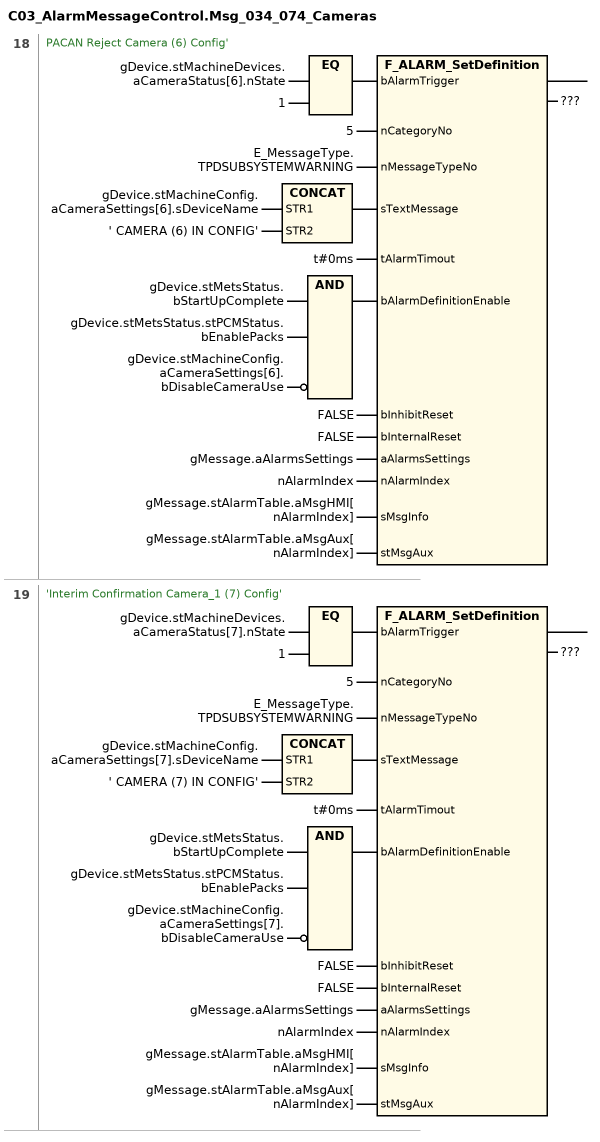
// NETWORK 18
// PACAN Reject Camera (6) Config'
F_ALARM_SetDefinition(bAlarmTrigger := gDevice.stMachineDevices.aCameraStatus[6].nState = 1, nCategoryNo := 5, nMessageTypeNo := E_MessageType.TPDSUBSYSTEMWARNING, sTextMessage := CONCAT(STR1 := gDevice.stMachineConfig.aCameraSettings[6].sDeviceName, STR2 := ' CAMERA (6) IN CONFIG'), tAlarmTimout := t#0ms, bAlarmDefinitionEnable := gDevice.stMetsStatus.bStartUpComplete AND gDevice.stMetsStatus.stPCMStatus.bEnablePacks AND NOT gDevice.stMachineConfig.aCameraSettings[6].bDisableCameraUse, bInhibitReset := FALSE, bInternalReset := FALSE, aAlarmsSettings := gMessage.aAlarmsSettings, nAlarmIndex := nAlarmIndex, sMsgInfo := gMessage.stAlarmTable.aMsgHMI[nAlarmIndex], stMsgAux := gMessage.stAlarmTable.aMsgAux[nAlarmIndex]);

// NETWORK 19
// 'Interim Confirmation Camera_1 (7) Config'
F_ALARM_SetDefinition(bAlarmTrigger := gDevice.stMachineDevices.aCameraStatus[7].nState = 1, nCategoryNo := 5, nMessageTypeNo := E_MessageType.TPDSUBSYSTEMWARNING, sTextMessage := CONCAT(STR1 := gDevice.stMachineConfig.aCameraSettings[7].sDeviceName, STR2 := ' CAMERA (7) IN CONFIG'), tAlarmTimout := t#0ms, bAlarmDefinitionEnable := gDevice.stMetsStatus.bStartUpComplete AND gDevice.stMetsStatus.stPCMStatus.bEnablePacks AND NOT gDevice.stMachineConfig.aCameraSettings[7].bDisableCameraUse, bInhibitReset := FALSE, bInternalReset := FALSE, aAlarmsSettings := gMessage.aAlarmsSettings, nAlarmIndex := nAlarmIndex, sMsgInfo := gMessage.stAlarmTable.aMsgHMI[nAlarmIndex], stMsgAux := gMessage.stAlarmTable.aMsgAux[nAlarmIndex]);

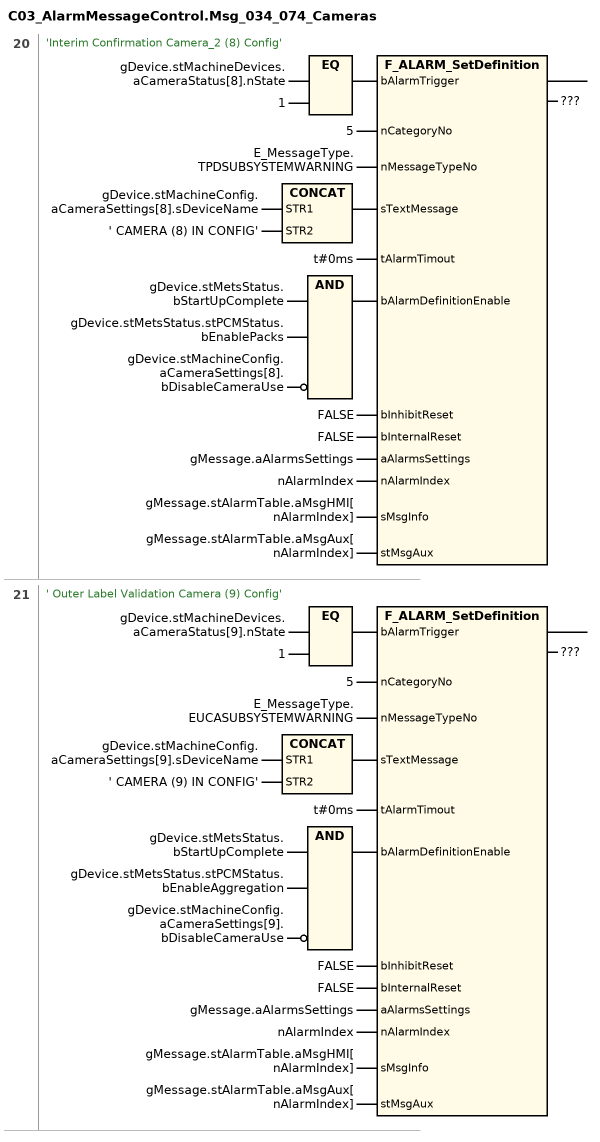
// NETWORK 20
// 'Interim Confirmation Camera_2 (8) Config'
F_ALARM_SetDefinition(bAlarmTrigger := gDevice.stMachineDevices.aCameraStatus[8].nState = 1, nCategoryNo := 5, nMessageTypeNo := E_MessageType.TPDSUBSYSTEMWARNING, sTextMessage := CONCAT(STR1 := gDevice.stMachineConfig.aCameraSettings[8].sDeviceName, STR2 := ' CAMERA (8) IN CONFIG'), tAlarmTimout := t#0ms, bAlarmDefinitionEnable := gDevice.stMetsStatus.bStartUpComplete AND gDevice.stMetsStatus.stPCMStatus.bEnablePacks AND NOT gDevice.stMachineConfig.aCameraSettings[8].bDisableCameraUse, bInhibitReset := FALSE, bInternalReset := FALSE, aAlarmsSettings := gMessage.aAlarmsSettings, nAlarmIndex := nAlarmIndex, sMsgInfo := gMessage.stAlarmTable.aMsgHMI[nAlarmIndex], stMsgAux := gMessage.stAlarmTable.aMsgAux[nAlarmIndex]);

// NETWORK 21
// ' Outer Label Validation Camera (9) Config'
F_ALARM_SetDefinition(bAlarmTrigger := gDevice.stMachineDevices.aCameraStatus[9].nState = 1, nCategoryNo := 5, nMessageTypeNo := E_MessageType.EUCASUBSYSTEMWARNING, sTextMessage := CONCAT(STR1 := gDevice.stMachineConfig.aCameraSettings[9].sDeviceName, STR2 := ' CAMERA (9) IN CONFIG'), tAlarmTimout := t#0ms, bAlarmDefinitionEnable := gDevice.stMetsStatus.bStartUpComplete AND gDevice.stMetsStatus.stPCMStatus.bEnableAggregation AND NOT gDevice.stMachineConfig.aCameraSettings[9].bDisableCameraUse, bInhibitReset := FALSE, bInternalReset := FALSE, aAlarmsSettings := gMessage.aAlarmsSettings, nAlarmIndex := nAlarmIndex, sMsgInfo := gMessage.stAlarmTable.aMsgHMI[nAlarmIndex], stMsgAux := gMessage.stAlarmTable.aMsgAux[nAlarmIndex]);

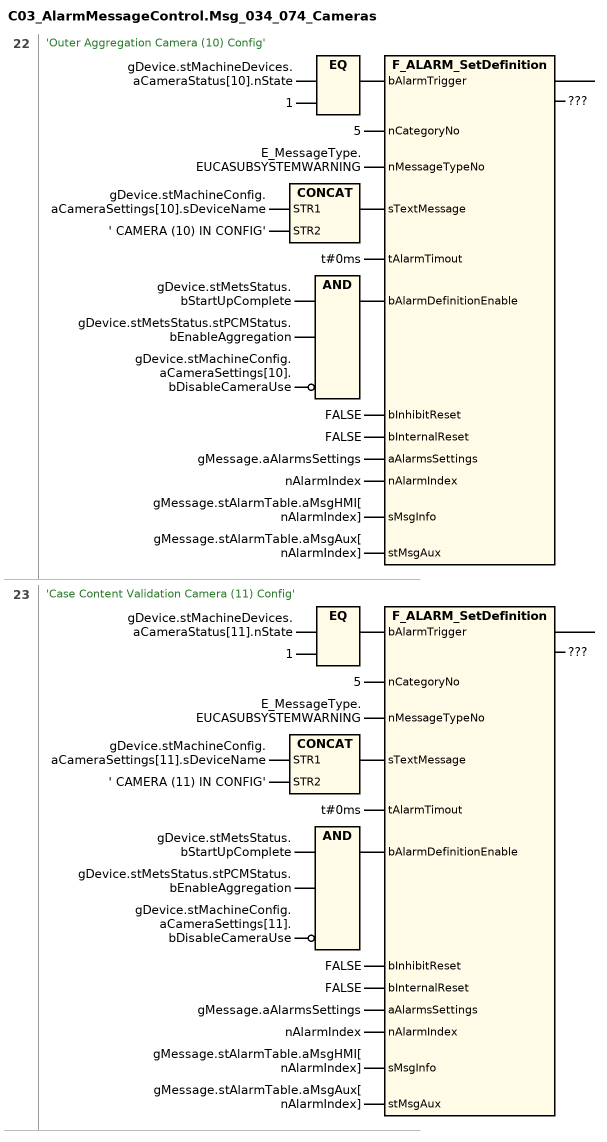
// NETWORK 22
// 'Outer Aggregation Camera (10) Config'
F_ALARM_SetDefinition(bAlarmTrigger := gDevice.stMachineDevices.aCameraStatus[10].nState = 1, nCategoryNo := 5, nMessageTypeNo := E_MessageType.EUCASUBSYSTEMWARNING, sTextMessage := CONCAT(STR1 := gDevice.stMachineConfig.aCameraSettings[10].sDeviceName, STR2 := ' CAMERA (10) IN CONFIG'), tAlarmTimout := t#0ms, bAlarmDefinitionEnable := gDevice.stMetsStatus.bStartUpComplete AND gDevice.stMetsStatus.stPCMStatus.bEnableAggregation AND NOT gDevice.stMachineConfig.aCameraSettings[10].bDisableCameraUse, bInhibitReset := FALSE, bInternalReset := FALSE, aAlarmsSettings := gMessage.aAlarmsSettings, nAlarmIndex := nAlarmIndex, sMsgInfo := gMessage.stAlarmTable.aMsgHMI[nAlarmIndex], stMsgAux := gMessage.stAlarmTable.aMsgAux[nAlarmIndex]);

// NETWORK 23
// 'Case Content Validation Camera (11) Config'
F_ALARM_SetDefinition(bAlarmTrigger := gDevice.stMachineDevices.aCameraStatus[11].nState = 1, nCategoryNo := 5, nMessageTypeNo := E_MessageType.EUCASUBSYSTEMWARNING, sTextMessage := CONCAT(STR1 := gDevice.stMachineConfig.aCameraSettings[11].sDeviceName, STR2 := ' CAMERA (11) IN CONFIG'), tAlarmTimout := t#0ms, bAlarmDefinitionEnable := gDevice.stMetsStatus.bStartUpComplete AND gDevice.stMetsStatus.stPCMStatus.bEnableAggregation AND NOT gDevice.stMachineConfig.aCameraSettings[11].bDisableCameraUse, bInhibitReset := FALSE, bInternalReset := FALSE, aAlarmsSettings := gMessage.aAlarmsSettings, nAlarmIndex := nAlarmIndex, sMsgInfo := gMessage.stAlarmTable.aMsgHMI[nAlarmIndex], stMsgAux := gMessage.stAlarmTable.aMsgAux[nAlarmIndex]);

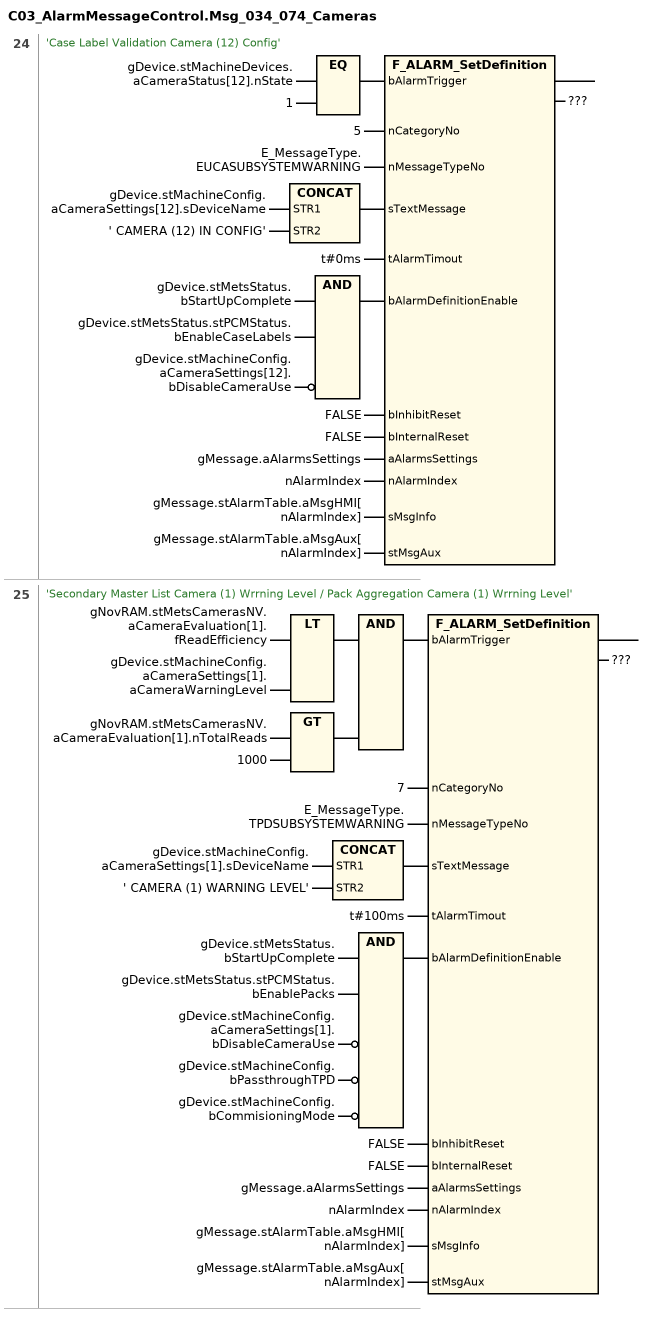
// NETWORK 24
// 'Case Label Validation Camera (12) Config'
F_ALARM_SetDefinition(bAlarmTrigger := gDevice.stMachineDevices.aCameraStatus[12].nState = 1, nCategoryNo := 5, nMessageTypeNo := E_MessageType.EUCASUBSYSTEMWARNING, sTextMessage := CONCAT(STR1 := gDevice.stMachineConfig.aCameraSettings[12].sDeviceName, STR2 := ' CAMERA (12) IN CONFIG'), tAlarmTimout := t#0ms, bAlarmDefinitionEnable := gDevice.stMetsStatus.bStartUpComplete AND gDevice.stMetsStatus.stPCMStatus.bEnableCaseLabels AND NOT gDevice.stMachineConfig.aCameraSettings[12].bDisableCameraUse, bInhibitReset := FALSE, bInternalReset := FALSE, aAlarmsSettings := gMessage.aAlarmsSettings, nAlarmIndex := nAlarmIndex, sMsgInfo := gMessage.stAlarmTable.aMsgHMI[nAlarmIndex], stMsgAux := gMessage.stAlarmTable.aMsgAux[nAlarmIndex]);

// NETWORK 25
// 'Secondary Master List Camera (1) Wrrning Level / Pack Aggregation Camera (1) Wrrning Level'
F_ALARM_SetDefinition(bAlarmTrigger := gNovRAM.stMetsCamerasNV.aCameraEvaluation[1].fReadEfficiency < gDevice.stMachineConfig.aCameraSettings[1].aCameraWarningLevel AND gNovRAM.stMetsCamerasNV.aCameraEvaluation[1].nTotalReads > 1000, nCategoryNo := 7, nMessageTypeNo := E_MessageType.TPDSUBSYSTEMWARNING, sTextMessage := CONCAT(STR1 := gDevice.stMachineConfig.aCameraSettings[1].sDeviceName, STR2 := ' CAMERA (1) WARNING LEVEL'), tAlarmTimout := t#100ms, bAlarmDefinitionEnable := gDevice.stMetsStatus.bStartUpComplete AND gDevice.stMetsStatus.stPCMStatus.bEnablePacks AND NOT gDevice.stMachineConfig.aCameraSettings[1].bDisableCameraUse AND NOT gDevice.stMachineConfig.bPassthroughTPD AND NOT gDevice.stMachineConfig.bCommisioningMode, bInhibitReset := FALSE, bInternalReset := FALSE, aAlarmsSettings := gMessage.aAlarmsSettings, nAlarmIndex := nAlarmIndex, sMsgInfo := gMessage.stAlarmTable.aMsgHMI[nAlarmIndex], stMsgAux := gMessage.stAlarmTable.aMsgAux[nAlarmIndex]);

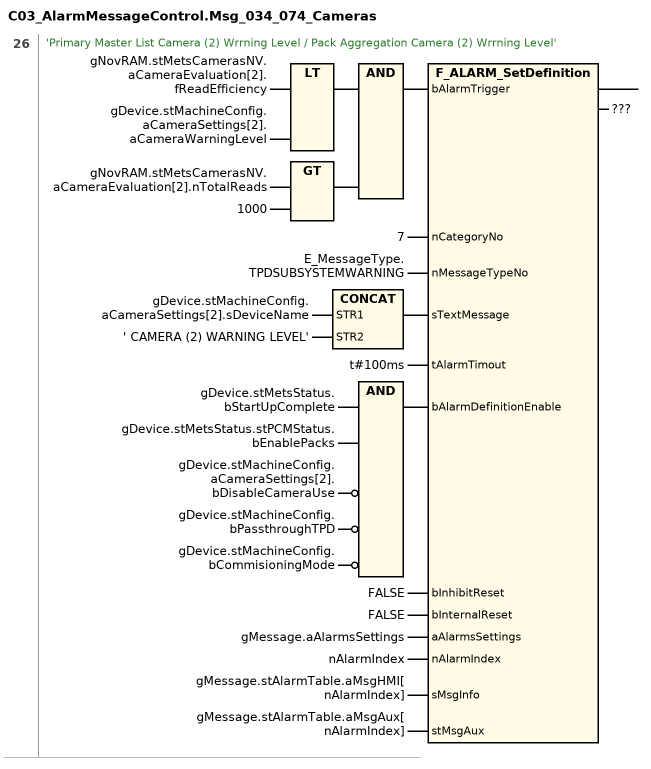
// NETWORK 26
// 'Primary Master List Camera (2) Wrrning Level / Pack Aggregation Camera (2) Wrrning Level'
F_ALARM_SetDefinition(bAlarmTrigger := gNovRAM.stMetsCamerasNV.aCameraEvaluation[2].fReadEfficiency < gDevice.stMachineConfig.aCameraSettings[2].aCameraWarningLevel AND gNovRAM.stMetsCamerasNV.aCameraEvaluation[2].nTotalReads > 1000, nCategoryNo := 7, nMessageTypeNo := E_MessageType.TPDSUBSYSTEMWARNING, sTextMessage := CONCAT(STR1 := gDevice.stMachineConfig.aCameraSettings[2].sDeviceName, STR2 := ' CAMERA (2) WARNING LEVEL'), tAlarmTimout := t#100ms, bAlarmDefinitionEnable := gDevice.stMetsStatus.bStartUpComplete AND gDevice.stMetsStatus.stPCMStatus.bEnablePacks AND NOT gDevice.stMachineConfig.aCameraSettings[2].bDisableCameraUse AND NOT gDevice.stMachineConfig.bPassthroughTPD AND NOT gDevice.stMachineConfig.bCommisioningMode, bInhibitReset := FALSE, bInternalReset := FALSE, aAlarmsSettings := gMessage.aAlarmsSettings, nAlarmIndex := nAlarmIndex, sMsgInfo := gMessage.stAlarmTable.aMsgHMI[nAlarmIndex], stMsgAux := gMessage.stAlarmTable.aMsgAux[nAlarmIndex]);

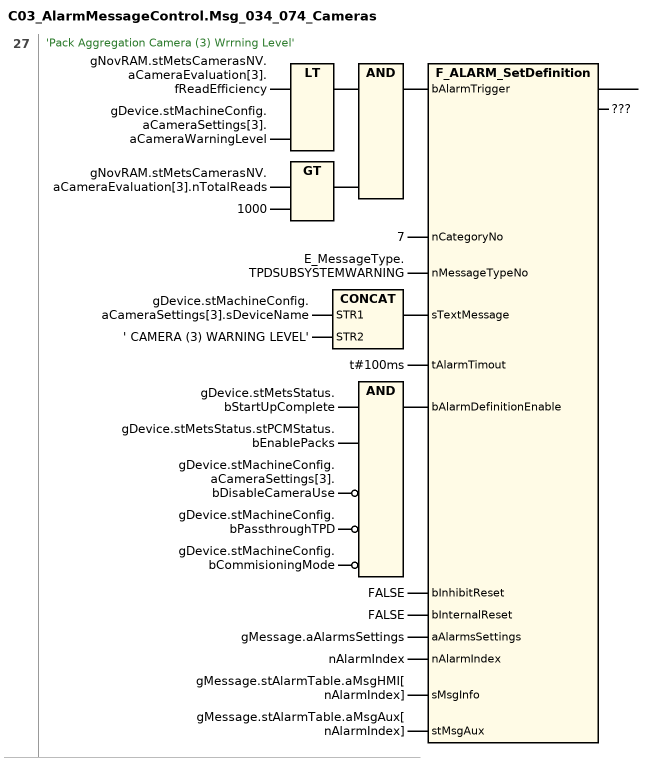
// NETWORK 27
// 'Pack Aggregation Camera (3) Wrrning Level'
F_ALARM_SetDefinition(bAlarmTrigger := gNovRAM.stMetsCamerasNV.aCameraEvaluation[3].fReadEfficiency < gDevice.stMachineConfig.aCameraSettings[3].aCameraWarningLevel AND gNovRAM.stMetsCamerasNV.aCameraEvaluation[3].nTotalReads > 1000, nCategoryNo := 7, nMessageTypeNo := E_MessageType.TPDSUBSYSTEMWARNING, sTextMessage := CONCAT(STR1 := gDevice.stMachineConfig.aCameraSettings[3].sDeviceName, STR2 := ' CAMERA (3) WARNING LEVEL'), tAlarmTimout := t#100ms, bAlarmDefinitionEnable := gDevice.stMetsStatus.bStartUpComplete AND gDevice.stMetsStatus.stPCMStatus.bEnablePacks AND NOT gDevice.stMachineConfig.aCameraSettings[3].bDisableCameraUse AND NOT gDevice.stMachineConfig.bPassthroughTPD AND NOT gDevice.stMachineConfig.bCommisioningMode, bInhibitReset := FALSE, bInternalReset := FALSE, aAlarmsSettings := gMessage.aAlarmsSettings, nAlarmIndex := nAlarmIndex, sMsgInfo := gMessage.stAlarmTable.aMsgHMI[nAlarmIndex], stMsgAux := gMessage.stAlarmTable.aMsgAux[nAlarmIndex]);

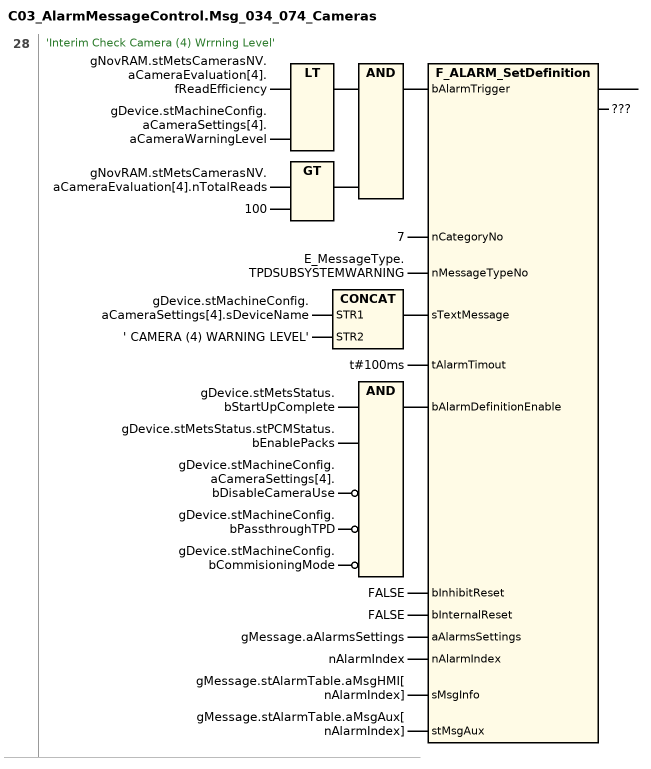
// NETWORK 28
// 'Interim Check Camera (4) Wrrning Level'
F_ALARM_SetDefinition(bAlarmTrigger := gNovRAM.stMetsCamerasNV.aCameraEvaluation[4].fReadEfficiency < gDevice.stMachineConfig.aCameraSettings[4].aCameraWarningLevel AND gNovRAM.stMetsCamerasNV.aCameraEvaluation[4].nTotalReads > 100, nCategoryNo := 7, nMessageTypeNo := E_MessageType.TPDSUBSYSTEMWARNING, sTextMessage := CONCAT(STR1 := gDevice.stMachineConfig.aCameraSettings[4].sDeviceName, STR2 := ' CAMERA (4) WARNING LEVEL'), tAlarmTimout := t#100ms, bAlarmDefinitionEnable := gDevice.stMetsStatus.bStartUpComplete AND gDevice.stMetsStatus.stPCMStatus.bEnablePacks AND NOT gDevice.stMachineConfig.aCameraSettings[4].bDisableCameraUse AND NOT gDevice.stMachineConfig.bPassthroughTPD AND NOT gDevice.stMachineConfig.bCommisioningMode, bInhibitReset := FALSE, bInternalReset := FALSE, aAlarmsSettings := gMessage.aAlarmsSettings, nAlarmIndex := nAlarmIndex, sMsgInfo := gMessage.stAlarmTable.aMsgHMI[nAlarmIndex], stMsgAux := gMessage.stAlarmTable.aMsgAux[nAlarmIndex]);

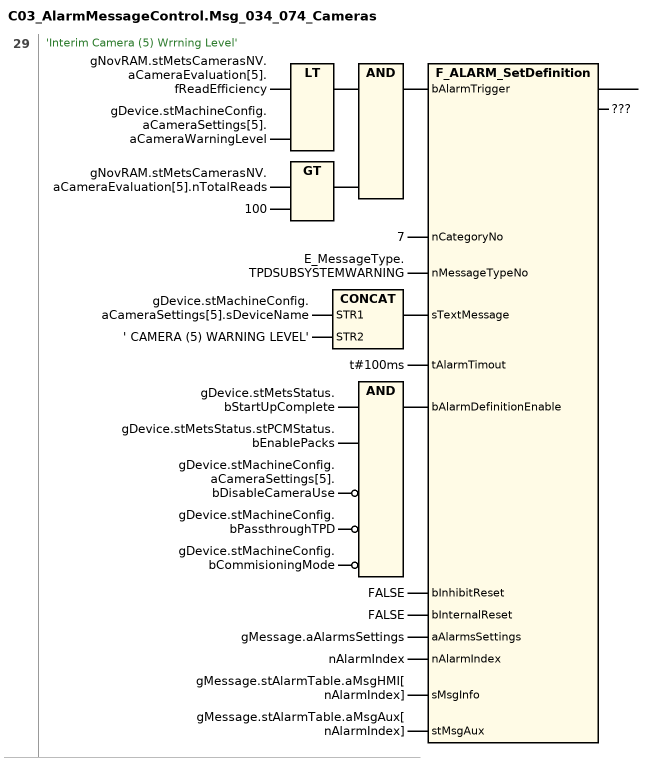
// NETWORK 29
// 'Interim Camera (5) Wrrning Level'
F_ALARM_SetDefinition(bAlarmTrigger := gNovRAM.stMetsCamerasNV.aCameraEvaluation[5].fReadEfficiency < gDevice.stMachineConfig.aCameraSettings[5].aCameraWarningLevel AND gNovRAM.stMetsCamerasNV.aCameraEvaluation[5].nTotalReads > 100, nCategoryNo := 7, nMessageTypeNo := E_MessageType.TPDSUBSYSTEMWARNING, sTextMessage := CONCAT(STR1 := gDevice.stMachineConfig.aCameraSettings[5].sDeviceName, STR2 := ' CAMERA (5) WARNING LEVEL'), tAlarmTimout := t#100ms, bAlarmDefinitionEnable := gDevice.stMetsStatus.bStartUpComplete AND gDevice.stMetsStatus.stPCMStatus.bEnablePacks AND NOT gDevice.stMachineConfig.aCameraSettings[5].bDisableCameraUse AND NOT gDevice.stMachineConfig.bPassthroughTPD AND NOT gDevice.stMachineConfig.bCommisioningMode, bInhibitReset := FALSE, bInternalReset := FALSE, aAlarmsSettings := gMessage.aAlarmsSettings, nAlarmIndex := nAlarmIndex, sMsgInfo := gMessage.stAlarmTable.aMsgHMI[nAlarmIndex], stMsgAux := gMessage.stAlarmTable.aMsgAux[nAlarmIndex]);

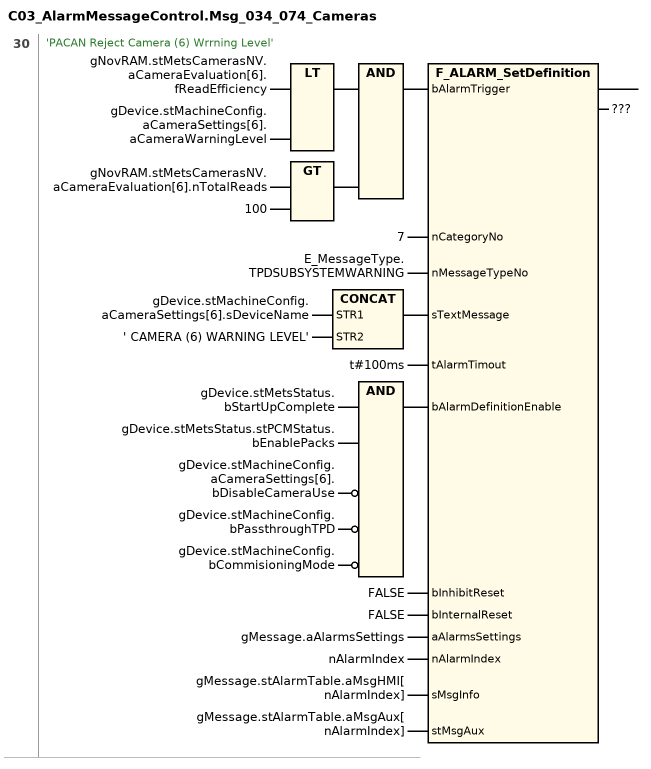
// NETWORK 30
// 'PACAN Reject Camera (6) Wrrning Level'
F_ALARM_SetDefinition(bAlarmTrigger := gNovRAM.stMetsCamerasNV.aCameraEvaluation[6].fReadEfficiency < gDevice.stMachineConfig.aCameraSettings[6].aCameraWarningLevel AND gNovRAM.stMetsCamerasNV.aCameraEvaluation[6].nTotalReads > 100, nCategoryNo := 7, nMessageTypeNo := E_MessageType.TPDSUBSYSTEMWARNING, sTextMessage := CONCAT(STR1 := gDevice.stMachineConfig.aCameraSettings[6].sDeviceName, STR2 := ' CAMERA (6) WARNING LEVEL'), tAlarmTimout := t#100ms, bAlarmDefinitionEnable := gDevice.stMetsStatus.bStartUpComplete AND gDevice.stMetsStatus.stPCMStatus.bEnablePacks AND NOT gDevice.stMachineConfig.aCameraSettings[6].bDisableCameraUse AND NOT gDevice.stMachineConfig.bPassthroughTPD AND NOT gDevice.stMachineConfig.bCommisioningMode, bInhibitReset := FALSE, bInternalReset := FALSE, aAlarmsSettings := gMessage.aAlarmsSettings, nAlarmIndex := nAlarmIndex, sMsgInfo := gMessage.stAlarmTable.aMsgHMI[nAlarmIndex], stMsgAux := gMessage.stAlarmTable.aMsgAux[nAlarmIndex]);

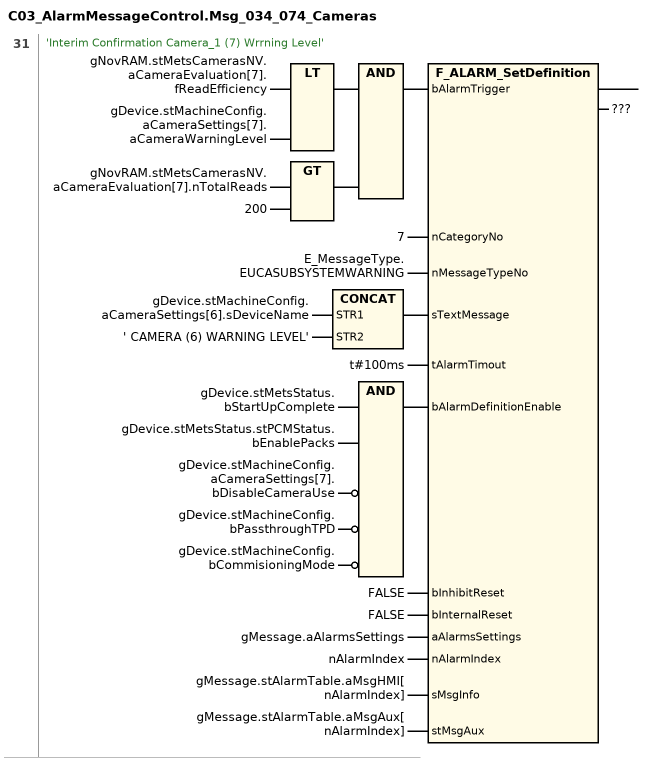
// NETWORK 31
// 'Interim Confirmation Camera_1 (7) Wrrning Level'
F_ALARM_SetDefinition(bAlarmTrigger := gNovRAM.stMetsCamerasNV.aCameraEvaluation[7].fReadEfficiency < gDevice.stMachineConfig.aCameraSettings[7].aCameraWarningLevel AND gNovRAM.stMetsCamerasNV.aCameraEvaluation[7].nTotalReads > 200, nCategoryNo := 7, nMessageTypeNo := E_MessageType.EUCASUBSYSTEMWARNING, sTextMessage := CONCAT(STR1 := gDevice.stMachineConfig.aCameraSettings[6].sDeviceName, STR2 := ' CAMERA (6) WARNING LEVEL'), tAlarmTimout := t#100ms, bAlarmDefinitionEnable := gDevice.stMetsStatus.bStartUpComplete AND gDevice.stMetsStatus.stPCMStatus.bEnablePacks AND NOT gDevice.stMachineConfig.aCameraSettings[7].bDisableCameraUse AND NOT gDevice.stMachineConfig.bPassthroughTPD AND NOT gDevice.stMachineConfig.bCommisioningMode, bInhibitReset := FALSE, bInternalReset := FALSE, aAlarmsSettings := gMessage.aAlarmsSettings, nAlarmIndex := nAlarmIndex, sMsgInfo := gMessage.stAlarmTable.aMsgHMI[nAlarmIndex], stMsgAux := gMessage.stAlarmTable.aMsgAux[nAlarmIndex]);

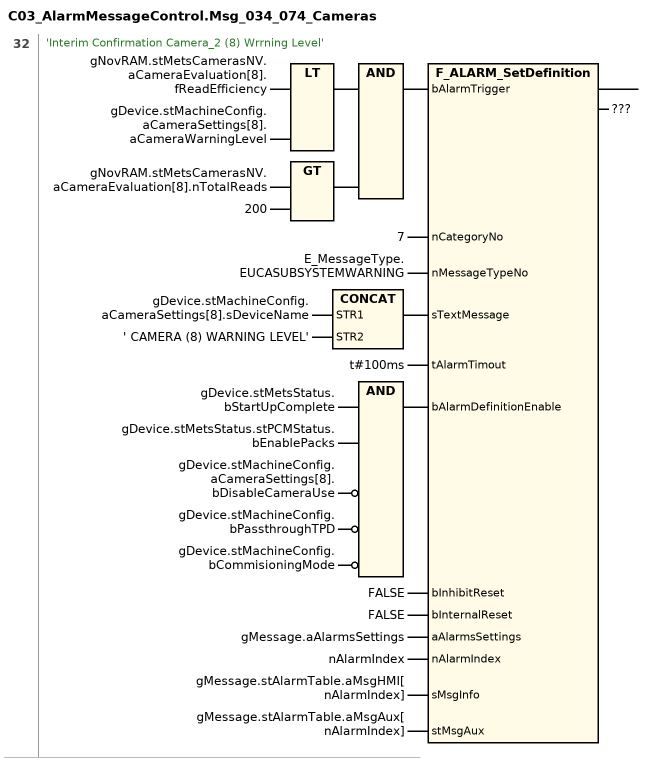
// NETWORK 32
// 'Interim Confirmation Camera_2 (8) Wrrning Level'
F_ALARM_SetDefinition(bAlarmTrigger := gNovRAM.stMetsCamerasNV.aCameraEvaluation[8].fReadEfficiency < gDevice.stMachineConfig.aCameraSettings[8].aCameraWarningLevel AND gNovRAM.stMetsCamerasNV.aCameraEvaluation[8].nTotalReads > 200, nCategoryNo := 7, nMessageTypeNo := E_MessageType.EUCASUBSYSTEMWARNING, sTextMessage := CONCAT(STR1 := gDevice.stMachineConfig.aCameraSettings[8].sDeviceName, STR2 := ' CAMERA (8) WARNING LEVEL'), tAlarmTimout := t#100ms, bAlarmDefinitionEnable := gDevice.stMetsStatus.bStartUpComplete AND gDevice.stMetsStatus.stPCMStatus.bEnablePacks AND NOT gDevice.stMachineConfig.aCameraSettings[8].bDisableCameraUse AND NOT gDevice.stMachineConfig.bPassthroughTPD AND NOT gDevice.stMachineConfig.bCommisioningMode, bInhibitReset := FALSE, bInternalReset := FALSE, aAlarmsSettings := gMessage.aAlarmsSettings, nAlarmIndex := nAlarmIndex, sMsgInfo := gMessage.stAlarmTable.aMsgHMI[nAlarmIndex], stMsgAux := gMessage.stAlarmTable.aMsgAux[nAlarmIndex]);

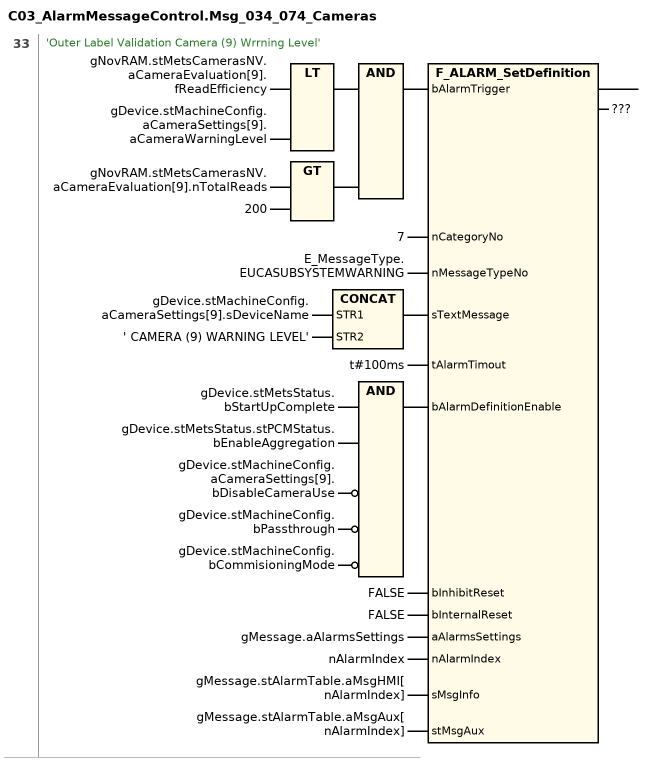
// NETWORK 33
// 'Outer Label Validation Camera (9) Wrrning Level'
F_ALARM_SetDefinition(bAlarmTrigger := gNovRAM.stMetsCamerasNV.aCameraEvaluation[9].fReadEfficiency < gDevice.stMachineConfig.aCameraSettings[9].aCameraWarningLevel AND gNovRAM.stMetsCamerasNV.aCameraEvaluation[9].nTotalReads > 200, nCategoryNo := 7, nMessageTypeNo := E_MessageType.EUCASUBSYSTEMWARNING, sTextMessage := CONCAT(STR1 := gDevice.stMachineConfig.aCameraSettings[9].sDeviceName, STR2 := ' CAMERA (9) WARNING LEVEL'), tAlarmTimout := t#100ms, bAlarmDefinitionEnable := gDevice.stMetsStatus.bStartUpComplete AND gDevice.stMetsStatus.stPCMStatus.bEnableAggregation AND NOT gDevice.stMachineConfig.aCameraSettings[9].bDisableCameraUse AND NOT gDevice.stMachineConfig.bPassthrough AND NOT gDevice.stMachineConfig.bCommisioningMode, bInhibitReset := FALSE, bInternalReset := FALSE, aAlarmsSettings := gMessage.aAlarmsSettings, nAlarmIndex := nAlarmIndex, sMsgInfo := gMessage.stAlarmTable.aMsgHMI[nAlarmIndex], stMsgAux := gMessage.stAlarmTable.aMsgAux[nAlarmIndex]);

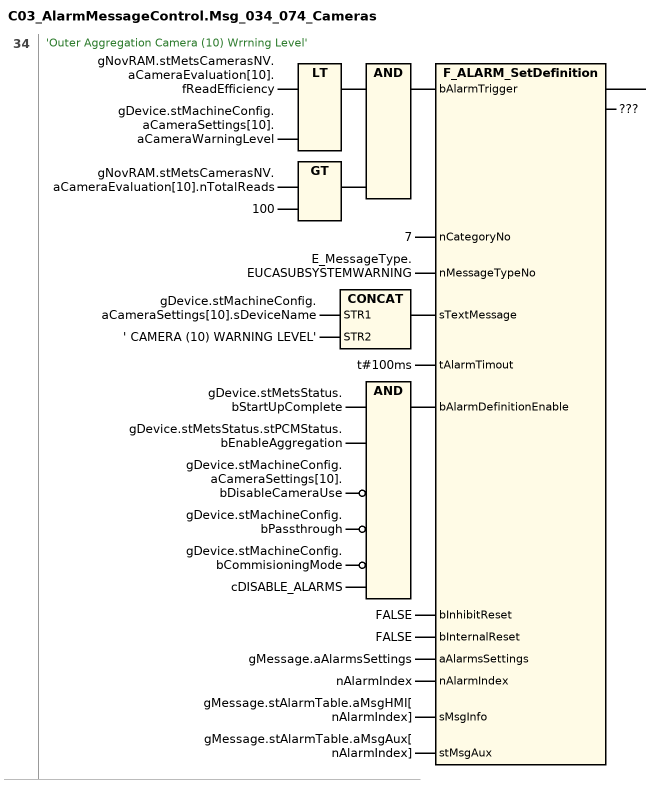
// NETWORK 34
// 'Outer Aggregation Camera (10) Wrrning Level'
F_ALARM_SetDefinition(bAlarmTrigger := gNovRAM.stMetsCamerasNV.aCameraEvaluation[10].fReadEfficiency < gDevice.stMachineConfig.aCameraSettings[10].aCameraWarningLevel AND gNovRAM.stMetsCamerasNV.aCameraEvaluation[10].nTotalReads > 100, nCategoryNo := 7, nMessageTypeNo := E_MessageType.EUCASUBSYSTEMWARNING, sTextMessage := CONCAT(STR1 := gDevice.stMachineConfig.aCameraSettings[10].sDeviceName, STR2 := ' CAMERA (10) WARNING LEVEL'), tAlarmTimout := t#100ms, bAlarmDefinitionEnable := gDevice.stMetsStatus.bStartUpComplete AND gDevice.stMetsStatus.stPCMStatus.bEnableAggregation AND NOT gDevice.stMachineConfig.aCameraSettings[10].bDisableCameraUse AND NOT gDevice.stMachineConfig.bPassthrough AND NOT gDevice.stMachineConfig.bCommisioningMode AND cDISABLE_ALARMS, bInhibitReset := FALSE, bInternalReset := FALSE, aAlarmsSettings := gMessage.aAlarmsSettings, nAlarmIndex := nAlarmIndex, sMsgInfo := gMessage.stAlarmTable.aMsgHMI[nAlarmIndex], stMsgAux := gMessage.stAlarmTable.aMsgAux[nAlarmIndex]);

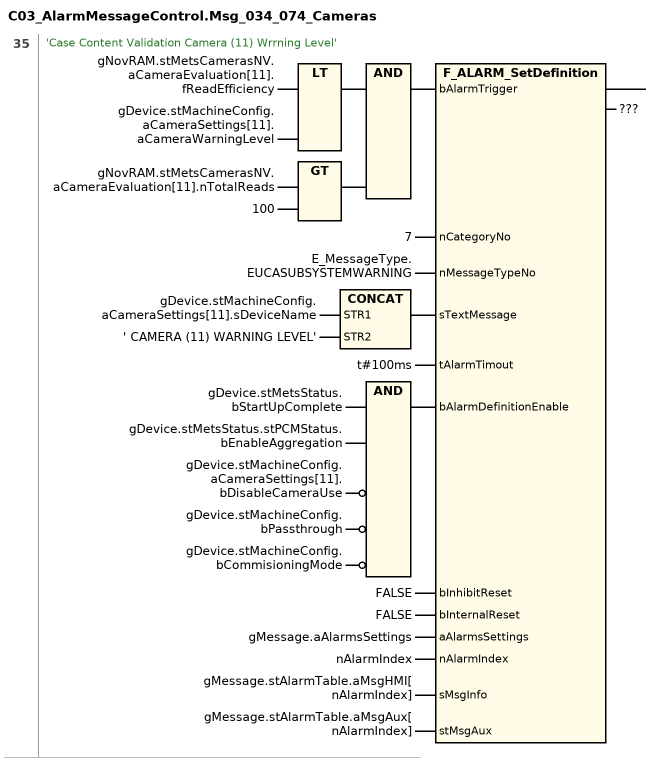
// NETWORK 35
// 'Case Content Validation Camera (11) Wrrning Level'
F_ALARM_SetDefinition(bAlarmTrigger := gNovRAM.stMetsCamerasNV.aCameraEvaluation[11].fReadEfficiency < gDevice.stMachineConfig.aCameraSettings[11].aCameraWarningLevel AND gNovRAM.stMetsCamerasNV.aCameraEvaluation[11].nTotalReads > 100, nCategoryNo := 7, nMessageTypeNo := E_MessageType.EUCASUBSYSTEMWARNING, sTextMessage := CONCAT(STR1 := gDevice.stMachineConfig.aCameraSettings[11].sDeviceName, STR2 := ' CAMERA (11) WARNING LEVEL'), tAlarmTimout := t#100ms, bAlarmDefinitionEnable := gDevice.stMetsStatus.bStartUpComplete AND gDevice.stMetsStatus.stPCMStatus.bEnableAggregation AND NOT gDevice.stMachineConfig.aCameraSettings[11].bDisableCameraUse AND NOT gDevice.stMachineConfig.bPassthrough AND NOT gDevice.stMachineConfig.bCommisioningMode, bInhibitReset := FALSE, bInternalReset := FALSE, aAlarmsSettings := gMessage.aAlarmsSettings, nAlarmIndex := nAlarmIndex, sMsgInfo := gMessage.stAlarmTable.aMsgHMI[nAlarmIndex], stMsgAux := gMessage.stAlarmTable.aMsgAux[nAlarmIndex]);

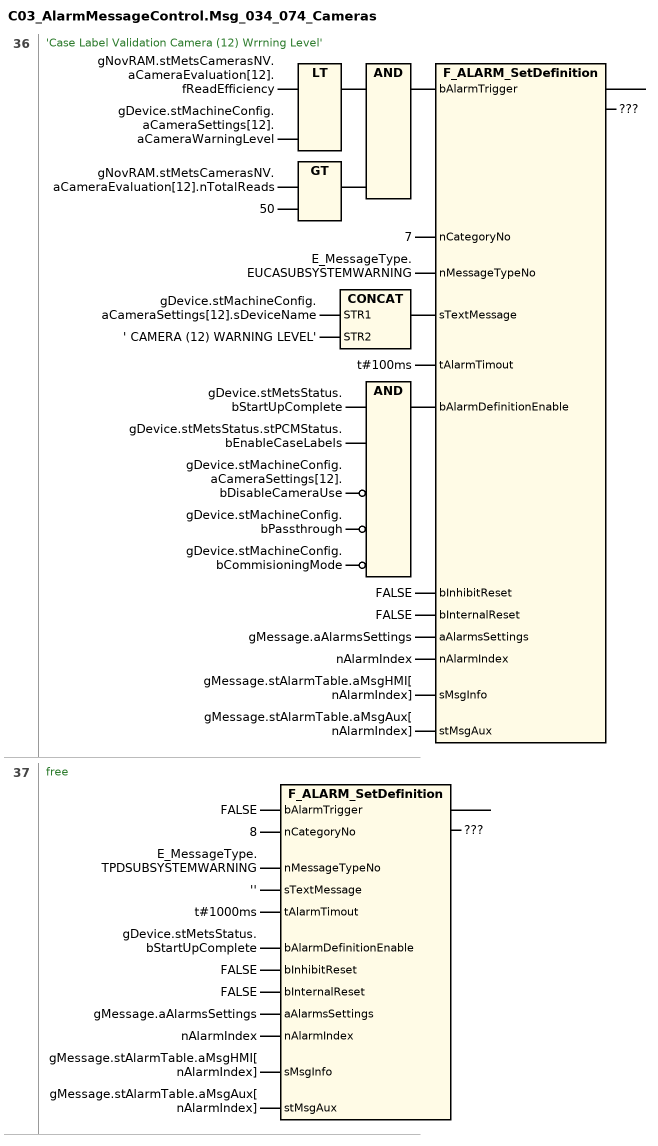
// NETWORK 36
// 'Case Label Validation Camera (12) Wrrning Level'
F_ALARM_SetDefinition(bAlarmTrigger := gNovRAM.stMetsCamerasNV.aCameraEvaluation[12].fReadEfficiency < gDevice.stMachineConfig.aCameraSettings[12].aCameraWarningLevel AND gNovRAM.stMetsCamerasNV.aCameraEvaluation[12].nTotalReads > 50, nCategoryNo := 7, nMessageTypeNo := E_MessageType.EUCASUBSYSTEMWARNING, sTextMessage := CONCAT(STR1 := gDevice.stMachineConfig.aCameraSettings[12].sDeviceName, STR2 := ' CAMERA (12) WARNING LEVEL'), tAlarmTimout := t#100ms, bAlarmDefinitionEnable := gDevice.stMetsStatus.bStartUpComplete AND gDevice.stMetsStatus.stPCMStatus.bEnableCaseLabels AND NOT gDevice.stMachineConfig.aCameraSettings[12].bDisableCameraUse AND NOT gDevice.stMachineConfig.bPassthrough AND NOT gDevice.stMachineConfig.bCommisioningMode, bInhibitReset := FALSE, bInternalReset := FALSE, aAlarmsSettings := gMessage.aAlarmsSettings, nAlarmIndex := nAlarmIndex, sMsgInfo := gMessage.stAlarmTable.aMsgHMI[nAlarmIndex], stMsgAux := gMessage.stAlarmTable.aMsgAux[nAlarmIndex]);

// NETWORK 37
// free
F_ALARM_SetDefinition(bAlarmTrigger := FALSE, nCategoryNo := 8, nMessageTypeNo := E_MessageType.TPDSUBSYSTEMWARNING, sTextMessage := '', tAlarmTimout := t#1000ms, bAlarmDefinitionEnable := gDevice.stMetsStatus.bStartUpComplete, bInhibitReset := FALSE, bInternalReset := FALSE, aAlarmsSettings := gMessage.aAlarmsSettings, nAlarmIndex := nAlarmIndex, sMsgInfo := gMessage.stAlarmTable.aMsgHMI[nAlarmIndex], stMsgAux := gMessage.stAlarmTable.aMsgAux[nAlarmIndex]);

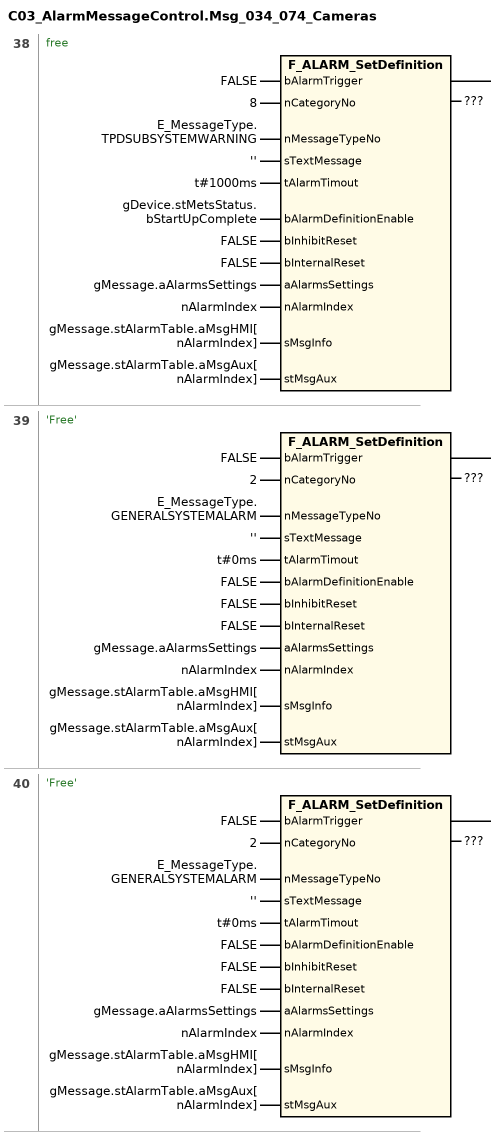
// NETWORK 38
// free
F_ALARM_SetDefinition(bAlarmTrigger := FALSE, nCategoryNo := 8, nMessageTypeNo := E_MessageType.TPDSUBSYSTEMWARNING, sTextMessage := '', tAlarmTimout := t#1000ms, bAlarmDefinitionEnable := gDevice.stMetsStatus.bStartUpComplete, bInhibitReset := FALSE, bInternalReset := FALSE, aAlarmsSettings := gMessage.aAlarmsSettings, nAlarmIndex := nAlarmIndex, sMsgInfo := gMessage.stAlarmTable.aMsgHMI[nAlarmIndex], stMsgAux := gMessage.stAlarmTable.aMsgAux[nAlarmIndex]);

// NETWORK 39
// 'Free'
F_ALARM_SetDefinition(bAlarmTrigger := FALSE, nCategoryNo := 2, nMessageTypeNo := E_MessageType.GENERALSYSTEMALARM, sTextMessage := '', tAlarmTimout := t#0ms, bAlarmDefinitionEnable := FALSE, bInhibitReset := FALSE, bInternalReset := FALSE, aAlarmsSettings := gMessage.aAlarmsSettings, nAlarmIndex := nAlarmIndex, sMsgInfo := gMessage.stAlarmTable.aMsgHMI[nAlarmIndex], stMsgAux := gMessage.stAlarmTable.aMsgAux[nAlarmIndex]);

// NETWORK 40
// 'Free'
F_ALARM_SetDefinition(bAlarmTrigger := FALSE, nCategoryNo := 2, nMessageTypeNo := E_MessageType.GENERALSYSTEMALARM, sTextMessage := '', tAlarmTimout := t#0ms, bAlarmDefinitionEnable := FALSE, bInhibitReset := FALSE, bInternalReset := FALSE, aAlarmsSettings := gMessage.aAlarmsSettings, nAlarmIndex := nAlarmIndex, sMsgInfo := gMessage.stAlarmTable.aMsgHMI[nAlarmIndex], stMsgAux := gMessage.stAlarmTable.aMsgAux[nAlarmIndex]);

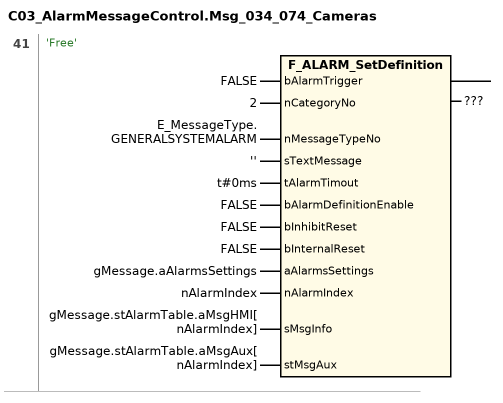
// NETWORK 41
// 'Free'
F_ALARM_SetDefinition(bAlarmTrigger := FALSE, nCategoryNo := 2, nMessageTypeNo := E_MessageType.GENERALSYSTEMALARM, sTextMessage := '', tAlarmTimout := t#0ms, bAlarmDefinitionEnable := FALSE, bInhibitReset := FALSE, bInternalReset := FALSE, aAlarmsSettings := gMessage.aAlarmsSettings, nAlarmIndex := nAlarmIndex, sMsgInfo := gMessage.stAlarmTable.aMsgHMI[nAlarmIndex], stMsgAux := gMessage.stAlarmTable.aMsgAux[nAlarmIndex]);
END_ACTION

ACTION Msg_075_126_Process:
// note: this text did not pass the execution check against the stored diagram
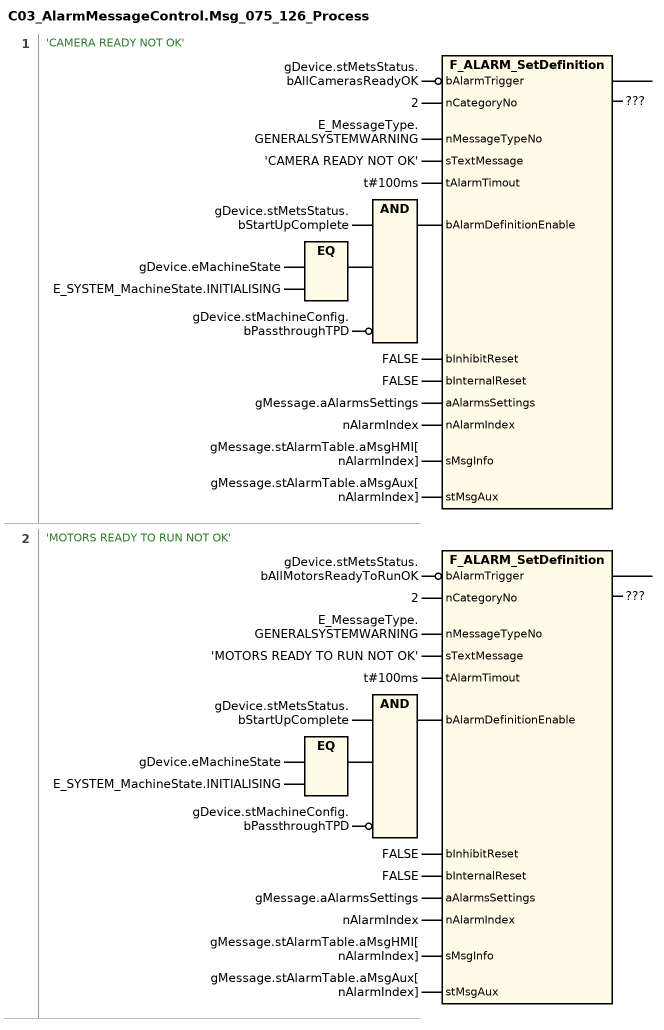
// NETWORK 1
// 'CAMERA READY NOT OK'
F_ALARM_SetDefinition(bAlarmTrigger := NOT gDevice.stMetsStatus.bAllCamerasReadyOK, nCategoryNo := 2, nMessageTypeNo := E_MessageType.GENERALSYSTEMWARNING, sTextMessage := 'CAMERA READY NOT OK', tAlarmTimout := t#100ms, bAlarmDefinitionEnable := gDevice.stMetsStatus.bStartUpComplete AND gDevice.eMachineState = E_SYSTEM_MachineState.INITIALISING AND NOT gDevice.stMachineConfig.bPassthroughTPD, bInhibitReset := FALSE, bInternalReset := FALSE, aAlarmsSettings := gMessage.aAlarmsSettings, nAlarmIndex := nAlarmIndex, sMsgInfo := gMessage.stAlarmTable.aMsgHMI[nAlarmIndex], stMsgAux := gMessage.stAlarmTable.aMsgAux[nAlarmIndex]);

// NETWORK 2
// 'MOTORS READY TO RUN NOT OK'
F_ALARM_SetDefinition(bAlarmTrigger := NOT gDevice.stMetsStatus.bAllMotorsReadyToRunOK, nCategoryNo := 2, nMessageTypeNo := E_MessageType.GENERALSYSTEMWARNING, sTextMessage := 'MOTORS READY TO RUN NOT OK', tAlarmTimout := t#100ms, bAlarmDefinitionEnable := gDevice.stMetsStatus.bStartUpComplete AND gDevice.eMachineState = E_SYSTEM_MachineState.INITIALISING AND NOT gDevice.stMachineConfig.bPassthroughTPD, bInhibitReset := FALSE, bInternalReset := FALSE, aAlarmsSettings := gMessage.aAlarmsSettings, nAlarmIndex := nAlarmIndex, sMsgInfo := gMessage.stAlarmTable.aMsgHMI[nAlarmIndex], stMsgAux := gMessage.stAlarmTable.aMsgAux[nAlarmIndex]);

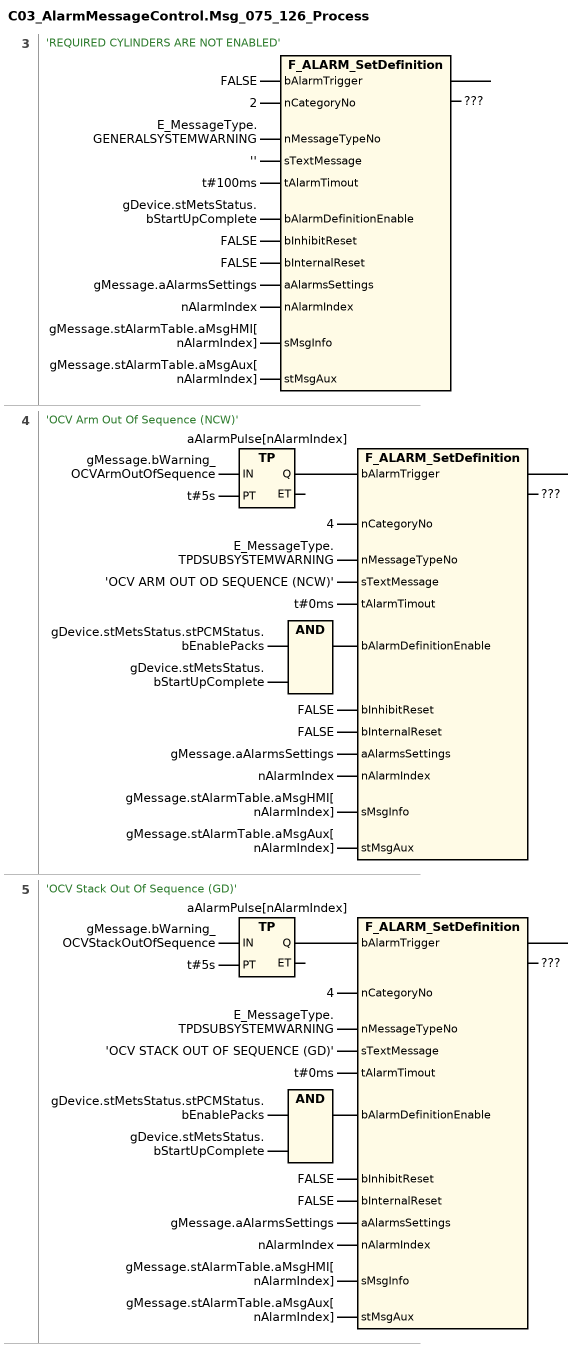
// NETWORK 3
// 'REQUIRED CYLINDERS ARE NOT ENABLED'
F_ALARM_SetDefinition(bAlarmTrigger := FALSE, nCategoryNo := 2, nMessageTypeNo := E_MessageType.GENERALSYSTEMWARNING, sTextMessage := '', tAlarmTimout := t#100ms, bAlarmDefinitionEnable := gDevice.stMetsStatus.bStartUpComplete, bInhibitReset := FALSE, bInternalReset := FALSE, aAlarmsSettings := gMessage.aAlarmsSettings, nAlarmIndex := nAlarmIndex, sMsgInfo := gMessage.stAlarmTable.aMsgHMI[nAlarmIndex], stMsgAux := gMessage.stAlarmTable.aMsgAux[nAlarmIndex]);

// NETWORK 4
// 'OCV Arm Out Of Sequence (NCW)'
aAlarmPulse[nAlarmIndex](IN := gMessage.bWarning_OCVArmOutOfSequence, PT := t#5s); // TP
F_ALARM_SetDefinition(bAlarmTrigger := aAlarmPulse[nAlarmIndex].Q, nCategoryNo := 4, nMessageTypeNo := E_MessageType.TPDSUBSYSTEMWARNING, sTextMessage := 'OCV ARM OUT OD SEQUENCE (NCW)', tAlarmTimout := t#0ms, bAlarmDefinitionEnable := gDevice.stMetsStatus.stPCMStatus.bEnablePacks AND gDevice.stMetsStatus.bStartUpComplete, bInhibitReset := FALSE, bInternalReset := FALSE, aAlarmsSettings := gMessage.aAlarmsSettings, nAlarmIndex := nAlarmIndex, sMsgInfo := gMessage.stAlarmTable.aMsgHMI[nAlarmIndex], stMsgAux := gMessage.stAlarmTable.aMsgAux[nAlarmIndex]);

// NETWORK 5
// 'OCV Stack Out Of Sequence (GD)'
aAlarmPulse[nAlarmIndex](IN := gMessage.bWarning_OCVStackOutOfSequence, PT := t#5s); // TP
F_ALARM_SetDefinition(bAlarmTrigger := aAlarmPulse[nAlarmIndex].Q, nCategoryNo := 4, nMessageTypeNo := E_MessageType.TPDSUBSYSTEMWARNING, sTextMessage := 'OCV STACK OUT OF SEQUENCE (GD)', tAlarmTimout := t#0ms, bAlarmDefinitionEnable := gDevice.stMetsStatus.stPCMStatus.bEnablePacks AND gDevice.stMetsStatus.bStartUpComplete, bInhibitReset := FALSE, bInternalReset := FALSE, aAlarmsSettings := gMessage.aAlarmsSettings, nAlarmIndex := nAlarmIndex, sMsgInfo := gMessage.stAlarmTable.aMsgHMI[nAlarmIndex], stMsgAux := gMessage.stAlarmTable.aMsgAux[nAlarmIndex]);

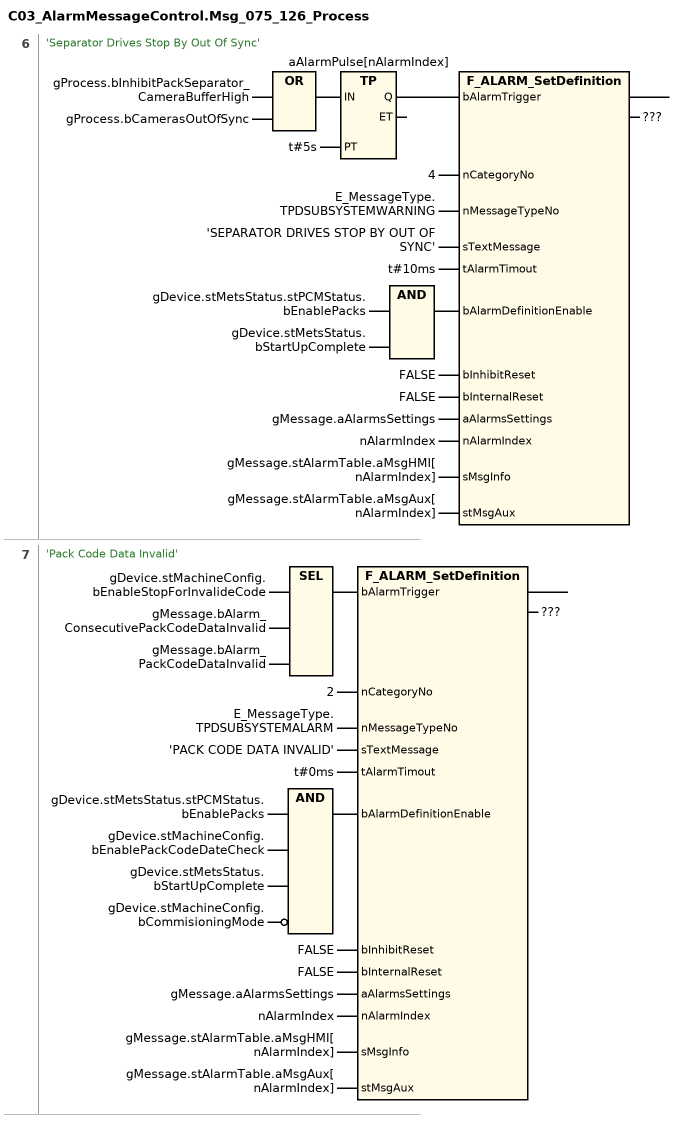
// NETWORK 6
// 'Separator Drives Stop By Out Of Sync'
aAlarmPulse[nAlarmIndex](IN := gProcess.bInhibitPackSeparator_CameraBufferHigh OR gProcess.bCamerasOutOfSync, PT := t#5s); // TP
F_ALARM_SetDefinition(bAlarmTrigger := aAlarmPulse[nAlarmIndex].Q, nCategoryNo := 4, nMessageTypeNo := E_MessageType.TPDSUBSYSTEMWARNING, sTextMessage := 'SEPARATOR DRIVES STOP BY OUT OF SYNC', tAlarmTimout := t#10ms, bAlarmDefinitionEnable := gDevice.stMetsStatus.stPCMStatus.bEnablePacks AND gDevice.stMetsStatus.bStartUpComplete, bInhibitReset := FALSE, bInternalReset := FALSE, aAlarmsSettings := gMessage.aAlarmsSettings, nAlarmIndex := nAlarmIndex, sMsgInfo := gMessage.stAlarmTable.aMsgHMI[nAlarmIndex], stMsgAux := gMessage.stAlarmTable.aMsgAux[nAlarmIndex]);

// NETWORK 7
// 'Pack Code Data Invalid'
F_ALARM_SetDefinition(bAlarmTrigger := SEL(gDevice.stMachineConfig.bEnableStopForInvalideCode, gMessage.bAlarm_ConsecutivePackCodeDataInvalid, gMessage.bAlarm_PackCodeDataInvalid), nCategoryNo := 2, nMessageTypeNo := E_MessageType.TPDSUBSYSTEMALARM, sTextMessage := 'PACK CODE DATA INVALID', tAlarmTimout := t#0ms, bAlarmDefinitionEnable := gDevice.stMetsStatus.stPCMStatus.bEnablePacks AND gDevice.stMachineConfig.bEnablePackCodeDateCheck AND gDevice.stMetsStatus.bStartUpComplete AND NOT gDevice.stMachineConfig.bCommisioningMode, bInhibitReset := FALSE, bInternalReset := FALSE, aAlarmsSettings := gMessage.aAlarmsSettings, nAlarmIndex := nAlarmIndex, sMsgInfo := gMessage.stAlarmTable.aMsgHMI[nAlarmIndex], stMsgAux := gMessage.stAlarmTable.aMsgAux[nAlarmIndex]);

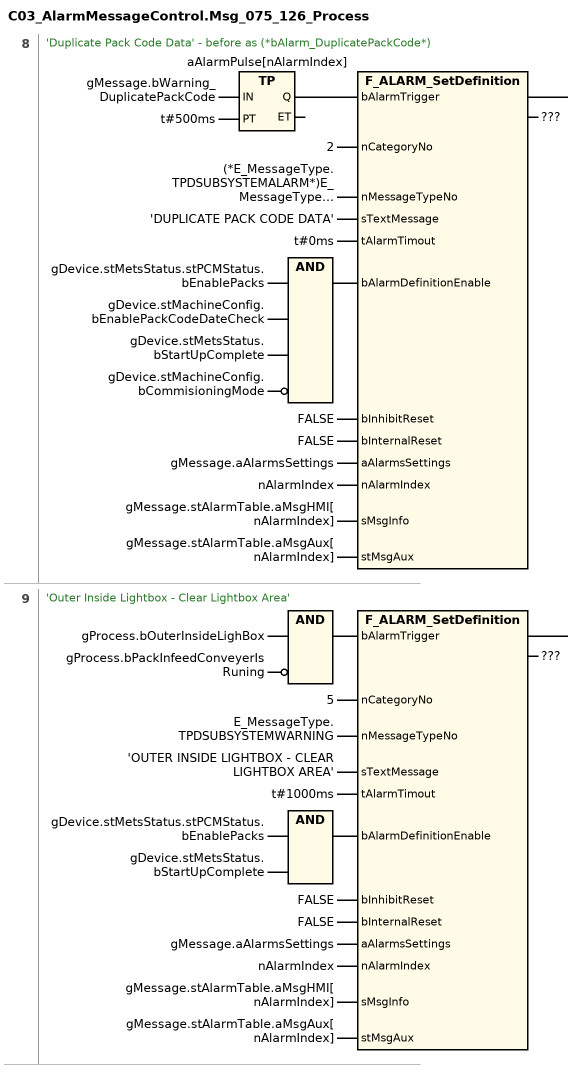
// NETWORK 8
// 'Duplicate Pack Code Data' - before as (*bAlarm_DuplicatePackCode*)
aAlarmPulse[nAlarmIndex](IN := gMessage.bWarning_DuplicatePackCode, PT := t#500ms); // TP
F_ALARM_SetDefinition(bAlarmTrigger := aAlarmPulse[nAlarmIndex].Q, nCategoryNo := 2, nMessageTypeNo := (*E_MessageType.TPDSUBSYSTEMALARM*)E_MessageType.TPDSUBSYSTEMWARNING, sTextMessage := 'DUPLICATE PACK CODE DATA', tAlarmTimout := t#0ms, bAlarmDefinitionEnable := gDevice.stMetsStatus.stPCMStatus.bEnablePacks AND gDevice.stMachineConfig.bEnablePackCodeDateCheck AND gDevice.stMetsStatus.bStartUpComplete AND NOT gDevice.stMachineConfig.bCommisioningMode, bInhibitReset := FALSE, bInternalReset := FALSE, aAlarmsSettings := gMessage.aAlarmsSettings, nAlarmIndex := nAlarmIndex, sMsgInfo := gMessage.stAlarmTable.aMsgHMI[nAlarmIndex], stMsgAux := gMessage.stAlarmTable.aMsgAux[nAlarmIndex]);

// NETWORK 9
// 'Outer Inside Lightbox - Clear Lightbox Area'
F_ALARM_SetDefinition(bAlarmTrigger := gProcess.bOuterInsideLighBox AND NOT gProcess.bPackInfeedConveyerIsRuning, nCategoryNo := 5, nMessageTypeNo := E_MessageType.TPDSUBSYSTEMWARNING, sTextMessage := 'OUTER INSIDE LIGHTBOX - CLEAR LIGHTBOX AREA', tAlarmTimout := t#1000ms, bAlarmDefinitionEnable := gDevice.stMetsStatus.stPCMStatus.bEnablePacks AND gDevice.stMetsStatus.bStartUpComplete, bInhibitReset := FALSE, bInternalReset := FALSE, aAlarmsSettings := gMessage.aAlarmsSettings, nAlarmIndex := nAlarmIndex, sMsgInfo := gMessage.stAlarmTable.aMsgHMI[nAlarmIndex], stMsgAux := gMessage.stAlarmTable.aMsgAux[nAlarmIndex]);

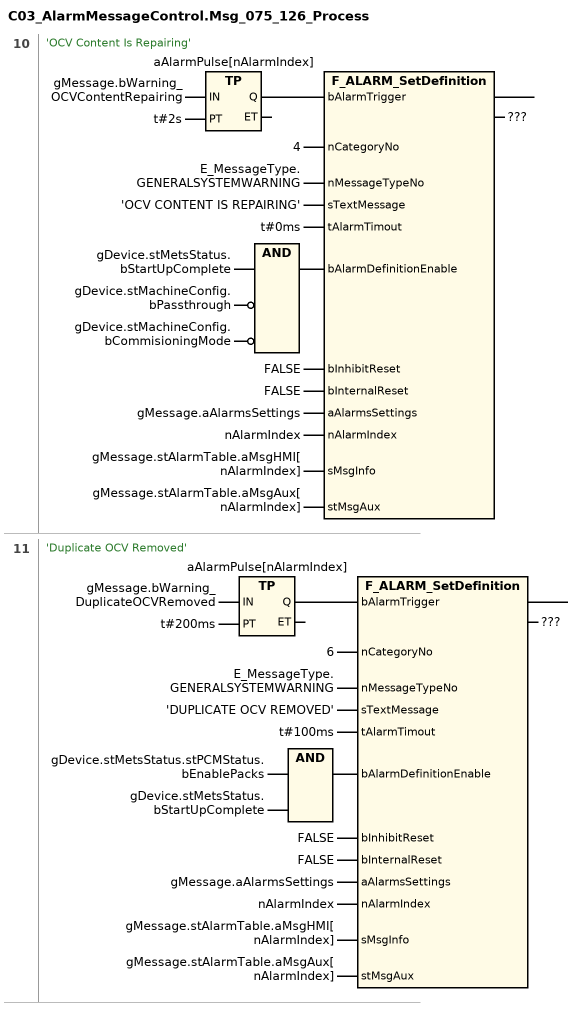
// NETWORK 10
// 'OCV Content Is Repairing'
aAlarmPulse[nAlarmIndex](IN := gMessage.bWarning_OCVContentRepairing, PT := t#2s); // TP
F_ALARM_SetDefinition(bAlarmTrigger := aAlarmPulse[nAlarmIndex].Q, nCategoryNo := 4, nMessageTypeNo := E_MessageType.GENERALSYSTEMWARNING, sTextMessage := 'OCV CONTENT IS REPAIRING', tAlarmTimout := t#0ms, bAlarmDefinitionEnable := gDevice.stMetsStatus.bStartUpComplete AND NOT gDevice.stMachineConfig.bPassthrough AND NOT gDevice.stMachineConfig.bCommisioningMode, bInhibitReset := FALSE, bInternalReset := FALSE, aAlarmsSettings := gMessage.aAlarmsSettings, nAlarmIndex := nAlarmIndex, sMsgInfo := gMessage.stAlarmTable.aMsgHMI[nAlarmIndex], stMsgAux := gMessage.stAlarmTable.aMsgAux[nAlarmIndex]);

// NETWORK 11
// 'Duplicate OCV Removed'
aAlarmPulse[nAlarmIndex](IN := gMessage.bWarning_DuplicateOCVRemoved, PT := t#200ms); // TP
F_ALARM_SetDefinition(bAlarmTrigger := aAlarmPulse[nAlarmIndex].Q, nCategoryNo := 6, nMessageTypeNo := E_MessageType.GENERALSYSTEMWARNING, sTextMessage := 'DUPLICATE OCV REMOVED', tAlarmTimout := t#100ms, bAlarmDefinitionEnable := gDevice.stMetsStatus.stPCMStatus.bEnablePacks AND gDevice.stMetsStatus.bStartUpComplete, bInhibitReset := FALSE, bInternalReset := FALSE, aAlarmsSettings := gMessage.aAlarmsSettings, nAlarmIndex := nAlarmIndex, sMsgInfo := gMessage.stAlarmTable.aMsgHMI[nAlarmIndex], stMsgAux := gMessage.stAlarmTable.aMsgAux[nAlarmIndex]);

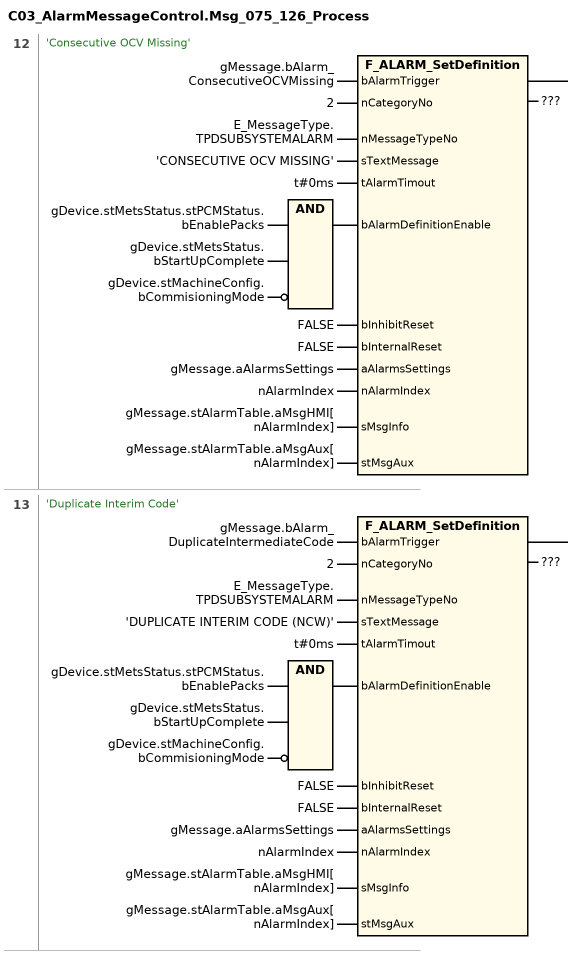
// NETWORK 12
// 'Consecutive OCV Missing'
F_ALARM_SetDefinition(bAlarmTrigger := gMessage.bAlarm_ConsecutiveOCVMissing, nCategoryNo := 2, nMessageTypeNo := E_MessageType.TPDSUBSYSTEMALARM, sTextMessage := 'CONSECUTIVE OCV MISSING', tAlarmTimout := t#0ms, bAlarmDefinitionEnable := gDevice.stMetsStatus.stPCMStatus.bEnablePacks AND gDevice.stMetsStatus.bStartUpComplete AND NOT gDevice.stMachineConfig.bCommisioningMode, bInhibitReset := FALSE, bInternalReset := FALSE, aAlarmsSettings := gMessage.aAlarmsSettings, nAlarmIndex := nAlarmIndex, sMsgInfo := gMessage.stAlarmTable.aMsgHMI[nAlarmIndex], stMsgAux := gMessage.stAlarmTable.aMsgAux[nAlarmIndex]);

// NETWORK 13
// 'Duplicate Interim Code'
F_ALARM_SetDefinition(bAlarmTrigger := gMessage.bAlarm_DuplicateIntermediateCode, nCategoryNo := 2, nMessageTypeNo := E_MessageType.TPDSUBSYSTEMALARM, sTextMessage := 'DUPLICATE INTERIM CODE (NCW)', tAlarmTimout := t#0ms, bAlarmDefinitionEnable := gDevice.stMetsStatus.stPCMStatus.bEnablePacks AND gDevice.stMetsStatus.bStartUpComplete AND NOT gDevice.stMachineConfig.bCommisioningMode, bInhibitReset := FALSE, bInternalReset := FALSE, aAlarmsSettings := gMessage.aAlarmsSettings, nAlarmIndex := nAlarmIndex, sMsgInfo := gMessage.stAlarmTable.aMsgHMI[nAlarmIndex], stMsgAux := gMessage.stAlarmTable.aMsgAux[nAlarmIndex]);

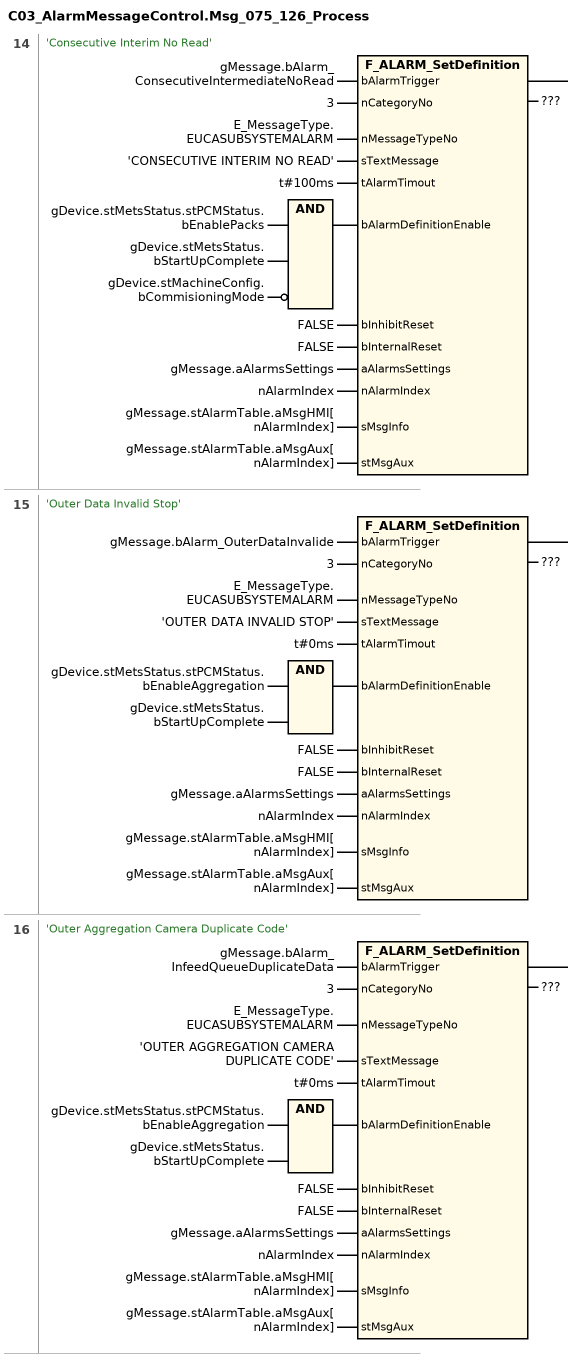
// NETWORK 14
// 'Consecutive Interim No Read'
F_ALARM_SetDefinition(bAlarmTrigger := gMessage.bAlarm_ConsecutiveIntermediateNoRead, nCategoryNo := 3, nMessageTypeNo := E_MessageType.EUCASUBSYSTEMALARM, sTextMessage := 'CONSECUTIVE INTERIM NO READ', tAlarmTimout := t#100ms, bAlarmDefinitionEnable := gDevice.stMetsStatus.stPCMStatus.bEnablePacks AND gDevice.stMetsStatus.bStartUpComplete AND NOT gDevice.stMachineConfig.bCommisioningMode, bInhibitReset := FALSE, bInternalReset := FALSE, aAlarmsSettings := gMessage.aAlarmsSettings, nAlarmIndex := nAlarmIndex, sMsgInfo := gMessage.stAlarmTable.aMsgHMI[nAlarmIndex], stMsgAux := gMessage.stAlarmTable.aMsgAux[nAlarmIndex]);

// NETWORK 15
// 'Outer Data Invalid Stop'
F_ALARM_SetDefinition(bAlarmTrigger := gMessage.bAlarm_OuterDataInvalide, nCategoryNo := 3, nMessageTypeNo := E_MessageType.EUCASUBSYSTEMALARM, sTextMessage := 'OUTER DATA INVALID STOP', tAlarmTimout := t#0ms, bAlarmDefinitionEnable := gDevice.stMetsStatus.stPCMStatus.bEnableAggregation AND gDevice.stMetsStatus.bStartUpComplete, bInhibitReset := FALSE, bInternalReset := FALSE, aAlarmsSettings := gMessage.aAlarmsSettings, nAlarmIndex := nAlarmIndex, sMsgInfo := gMessage.stAlarmTable.aMsgHMI[nAlarmIndex], stMsgAux := gMessage.stAlarmTable.aMsgAux[nAlarmIndex]);

// NETWORK 16
// 'Outer Aggregation Camera Duplicate Code'
F_ALARM_SetDefinition(bAlarmTrigger := gMessage.bAlarm_InfeedQueueDuplicateData, nCategoryNo := 3, nMessageTypeNo := E_MessageType.EUCASUBSYSTEMALARM, sTextMessage := 'OUTER AGGREGATION CAMERA DUPLICATE CODE', tAlarmTimout := t#0ms, bAlarmDefinitionEnable := gDevice.stMetsStatus.stPCMStatus.bEnableAggregation AND gDevice.stMetsStatus.bStartUpComplete, bInhibitReset := FALSE, bInternalReset := FALSE, aAlarmsSettings := gMessage.aAlarmsSettings, nAlarmIndex := nAlarmIndex, sMsgInfo := gMessage.stAlarmTable.aMsgHMI[nAlarmIndex], stMsgAux := gMessage.stAlarmTable.aMsgAux[nAlarmIndex]);

